{attribute 'GeneratedUsingTerminal: EL3751-0000-0020'}
{attribute addProperty BoxType "EL3751-0000-0020"}
{attribute addProperty Id "SamplesAT %I*Samples_F24E104A4"}
{attribute addProperty CRC "4003796773"}
{attribute addProperty Size "4"}
TYPE PAI_Samples_EEA51725 EXTENDS InputBase_8311D824 :
STRUCT
	{attribute addProperty Name "Samples"}
	Samples AT %I* : Samples_F24E104A;
END_STRUCT
END_TYPE

(* stored: Version 1.2.0.0, ProductVersion 3.1.4024.9
   DUT PAI_Samples_EEA51725: Id {2d4cfe63-6de5-4c8c-8e23-ea139814dce4} *)
